{attribute 'qualified_only'}
{attribute 'strict'}
TYPE E_Xts_StateMachine :
(
	enum_member := 0,
	Enabled := 1
);
END_TYPE

(* stored: Version 1.1.0.1, ProductVersion 3.1.4024.9
   DUT E_Xts_StateMachine: Id {9bb19fcb-a54b-4547-aaef-ae4667d753ae} *)
